% RSLogix 500 project cyclical_shift.RSS, saved by version 8.30.00.16 %
PROJECT "UNTITLED"    % processor: Bul.1763 MicroLogix 1100 Series B %

PROGRAM FILES
  LAD 2   4 rungs

DATA FILES
  O0 OUTPUT  4 elements
  I1 INPUT  6 elements
  S2 STATUS  66 elements
  B3 BINARY  1 elements
  T4 TIMER  1 elements
  C5 COUNTER  1 elements
  R6 CONTROL  1 elements
  N7 INTEGER  1 elements
  F8 FLOAT  1 elements
  N9 FIFO_PLUS1  6 elements

LADDER 2
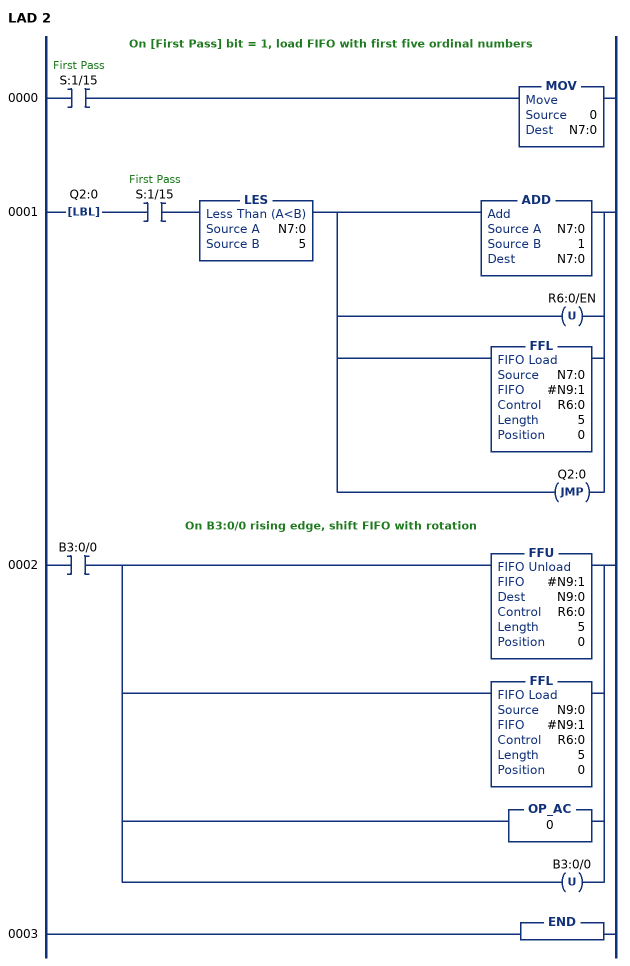
% Rung: 0 %
% TITLE: On [First Pass] bit = 1, load FIFO with first five ordinal numbers %
SOR XIC S:1/15 MOV 0 N7:0 EOR
%   S:1/15  "First Pass" %
% Rung: 1 %
SOR LBL Q2:0 XIC S:1/15 LES N7:0 5 BST ADD N7:0 1 N7:0 NXB OTU R6:0/EN NXB FFL N7:0 #N9:1 R6:0 5 0 NXB JMP Q2:0 BND EOR
%   S:1/15  "First Pass" %
% Rung: 2 %
% TITLE: On B3:0/0 rising edge, shift FIFO with rotation %
SOR XIC B3:0/0 BST FFU #N9:1 N9:0 R6:0 5 0 NXB FFL N9:0 #N9:1 R6:0 5 0 NXB OP_AC 0 NXB OTU B3:0/0 BND EOR
% Rung: 3 %
SOR END EOR

DATA TABLE (non-zero values as saved)
DATA R6
% .LEN .POS %
% R6:0 % 5 0
